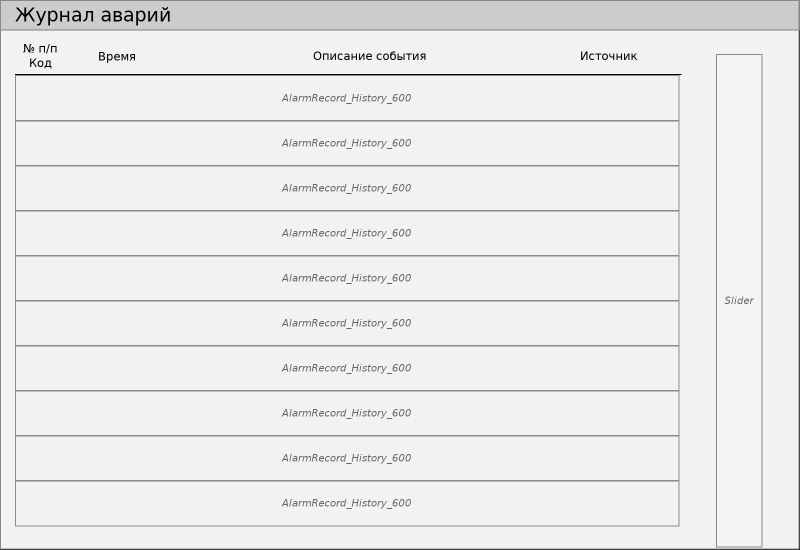
VISUALIZATION History_Of_Alarms_800x550  // 800x550
    Rectangle (0,0 800x550)
    Frame (15,75 664x46)
        shows AlarmRecord_History_600(AlarmRecord := PRG_Alarms_Core.HMI_HistoryAlarms[1], RecNum := PRG_Alarms_Core.HMI_NumsHY[1])
    Frame (15,120 664x46)
        shows AlarmRecord_History_600(AlarmRecord := PRG_Alarms_Core.HMI_HistoryAlarms[2], RecNum := PRG_Alarms_Core.HMI_NumsHY[2])
    Frame (15,165 664x46)
        shows AlarmRecord_History_600(AlarmRecord := PRG_Alarms_Core.HMI_HistoryAlarms[3], RecNum := PRG_Alarms_Core.HMI_NumsHY[3])
    Frame (15,210 664x46)
        shows AlarmRecord_History_600(AlarmRecord := PRG_Alarms_Core.HMI_HistoryAlarms[4], RecNum := PRG_Alarms_Core.HMI_NumsHY[4])
    Frame (15,255 664x46)
        shows AlarmRecord_History_600(AlarmRecord := PRG_Alarms_Core.HMI_HistoryAlarms[5], RecNum := PRG_Alarms_Core.HMI_NumsHY[5])
    Frame (15,300 664x46)
        shows AlarmRecord_History_600(AlarmRecord := PRG_Alarms_Core.HMI_HistoryAlarms[6], RecNum := PRG_Alarms_Core.HMI_NumsHY[6])
    Frame (15,345 664x46)
        shows AlarmRecord_History_600(AlarmRecord := PRG_Alarms_Core.HMI_HistoryAlarms[7], RecNum := PRG_Alarms_Core.HMI_NumsHY[7])
    Frame (15,390 664x46)
        shows AlarmRecord_History_600(AlarmRecord := PRG_Alarms_Core.HMI_HistoryAlarms[8], RecNum := PRG_Alarms_Core.HMI_NumsHY[8])
    Frame (15,435 664x46)
        shows AlarmRecord_History_600(AlarmRecord := PRG_Alarms_Core.HMI_HistoryAlarms[9], RecNum := PRG_Alarms_Core.HMI_NumsHY[9])
    Frame (15,480 664x46)
        shows AlarmRecord_History_600(AlarmRecord := PRG_Alarms_Core.HMI_HistoryAlarms[10], RecNum := PRG_Alarms_Core.HMI_NumsHY[10])
    Slider (716,54 46x493), variable: PRG_Alarms_Core.HMI_CurShiftHY, scale 0..1000
    Label (17,41 47x30), "№ п/п Код"
    Label (310,41 216x30), "Описание события"
    Label (577,41 77x30), "Источник"
    Label (91,47 52x19), "Время"
    Line (15,74) (681,74)
    Rectangle (0,0 800x30), "Журнал аварий"
END_VISUALIZATION

(* stored: Version 1.1.0.1, ProductVersion 3.1.4024.9
   Visu History_Of_Alarms_800x550: Id {e836338b-5b3a-4843-88a0-e28f9b26dbcf} *)
